FUNCTION_BLOCK Actuator_Transform (* Basic FB with empty ECC *)
  (* Standard: 61499-2 *)
  (* Version 1.0, 2023-03-02, AK125171 *)
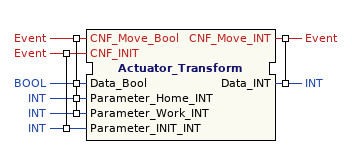
  EVENT_INPUT
    CNF_Move_Bool WITH Data_Bool, Parameter_Home_INT, Parameter_Work_INT;
    CNF_INIT WITH Parameter_INIT_INT;
  END_EVENT
  EVENT_OUTPUT
    CNF_Move_INT WITH Data_INT;
  END_EVENT
  VAR_INPUT
    Data_Bool : BOOL;
    Parameter_Home_INT : INT;
    Parameter_Work_INT : INT;
    Parameter_INIT_INT : INT;
  END_VAR
  VAR_OUTPUT
    Data_INT : INT;
  END_VAR
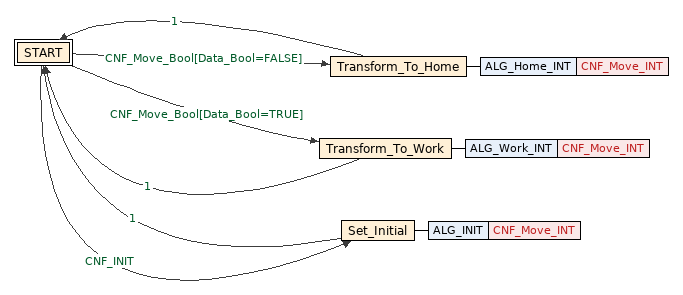
  EC_STATES
    START; (* Initial State *)
    Transform_To_Home : ALG_Home_INT -> CNF_Move_INT;
    Transform_To_Work : ALG_Work_INT -> CNF_Move_INT;
    Set_Initial : ALG_INIT -> CNF_Move_INT;
  END_STATES
  EC_TRANSITIONS
    START TO Transform_To_Home := CNF_Move_Bool[Data_Bool=FALSE];
    START TO Transform_To_Work := CNF_Move_Bool[Data_Bool=TRUE];
    Transform_To_Work TO START := 1;
    Transform_To_Home TO START := 1;
    START TO Set_Initial := CNF_INIT;
    Set_Initial TO START := 1;
  END_TRANSITIONS
  ALGORITHM ALG_Home_INT IN ST:
Data_INT:=Parameter_Home_INT;
  END_ALGORITHM
  ALGORITHM ALG_Work_INT IN ST:
Data_INT:=Parameter_Work_INT;
  END_ALGORITHM
  ALGORITHM ALG_INIT IN ST:
Data_INT:=Parameter_INIT_INT;
  END_ALGORITHM
END_FUNCTION_BLOCK
